Staubli VAL3: _WaitEnd.pgx

public program _WaitEnd()
// Halt robot here if "END" is activated
  local num nStateWaitEnd
begin
  // WAIT END OF CYCLE......................................................
  if SYS:CE_Requested and !SYS:bPartMade[moduleIndex] and SYS:doStartMachine[moduleIndex]==false
    do
      // Robot is running in production cycle (StateRobot==10)
      if SYS:nStateRobot==10 and isPowered() and SYS:diMachineInAuto[moduleIndex]==true
        // "End Of Cycle" running and no more parts in mould
        if SYS:CE_Requested and !SYS:bPartMade[moduleIndex] and SYS:diMachineInAuto[moduleIndex]==true
          nStateWaitEnd=30
        endIf
        // Robot Off called
        if SYS:bRobotOffCalled[moduleIndex]
          nStateWaitEnd=40
        endIf
      else
        // Robot or Machine not in AUTO
        if SYS:nStateRobot!=10
          nStateWaitEnd=0
        else
          // "End Of Cycle" running and no more parts in mould
          if SYS:CE_Requested and !SYS:bPartMade[moduleIndex] and SYS:CE_AtEndPos==false
            nStateWaitEnd=30
          endIf
          // Robot Off called
          if SYS:bRobotOffCalled[moduleIndex] and !bAtWaitPosition
            nStateWaitEnd=40
          endIf
        endIf
      endIf
      //
      switch (nStateWaitEnd)
        //
        //  Robot and Machine not in Auto.......................................
        case 0
          if SYS:diMachineInAuto[moduleIndex]==false
            //Wait Machine In Auto
            //user:sMessage[0]=user:sMessage[0]
          else
            //Wait [START] Robot
            //user:sMessage[0]=user:sMessage[0]
          endIf
        break
        //
        // "End Of Cycle" called and no more parts in mould.....................
        case 30
          if SYS:CE_Requested==true and SYS:bPartMade[moduleIndex]==false
            stopMove()
            wait(isSettled())
            SYS:CE_AtEndPos=true
            delay(0)
          endIf
        break
        //
        // Robot Off called.......................................................
        case 40
          wait(isSettled())
          stopMove()
          bAtWaitPosition=true
          delay(0)
        break
      endSwitch
      //
      // Wait until robot is at end position......................................
    until (SYS:CE_AtEndPos==true or bAtWaitPosition==true and isSettled())
    //
    // Reset StartMachine.................................................................................................
    SYS:doStartMachine[moduleIndex]=false
  endIf
end
